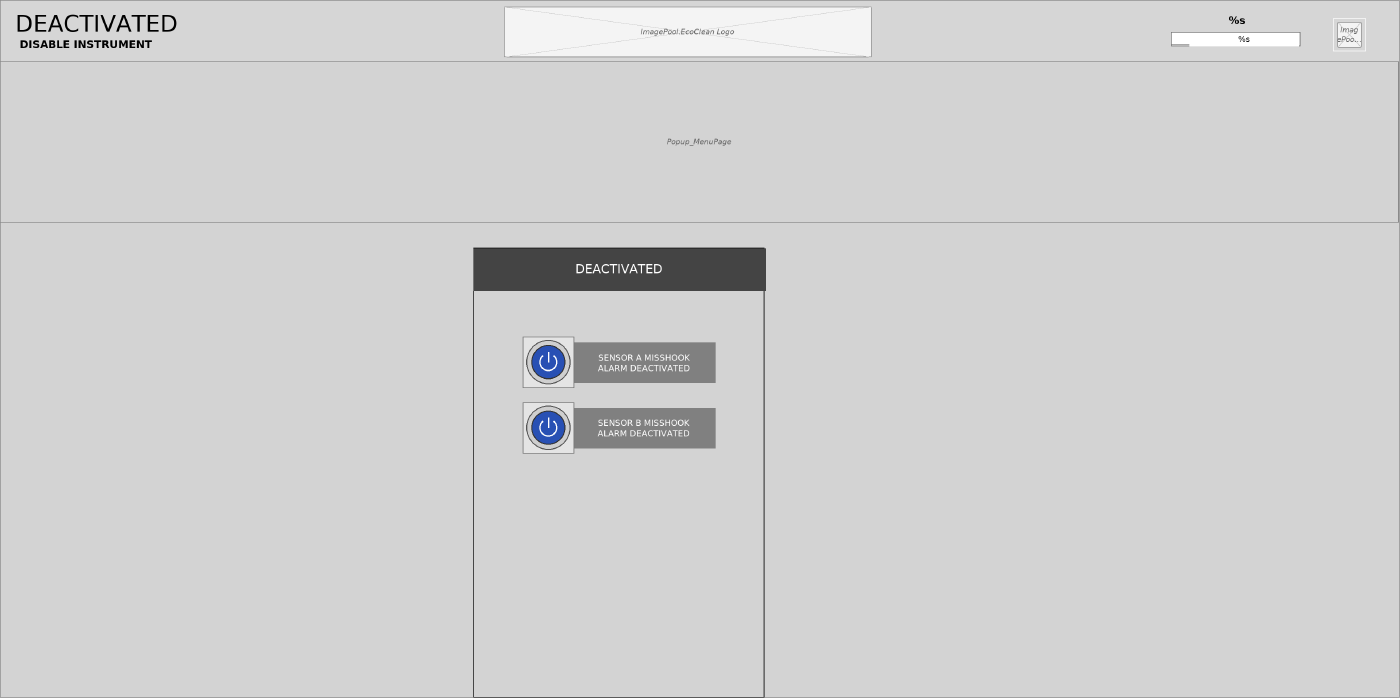
VISUALIZATION Deactivated_Page  // 1920x958
    Rectangle (0,63 1920x26)
        p3528305787: HMI_Ctrl.ANIMATION3
    Rectangle (0,0 1919x85)
    Label (18,6 267x53), "DEACTIVATED"
    Label (24,49 320x24), "DISABLE INSTRUMENT"
    Frame (0,84 1918x221), invisible if: HMI_Ctrl.CloseMenuButton
        shows Popup_MenuPage()
    Group (1828,25 45x45)
        OnMouseClick: toggle HMI_Ctrl.MenuButton
        RoundedRectangle (0,0 45x45), colour toggle: HMI_Ctrl.MenuButton
        Image (6,5 33x35), image: ImagePool.Menu Button
    Rectangle (649,340 399x618)
    Rectangle (649,341 401x58)
    Label (786,357 274x24), "DEACTIVATED"
    RoundedRectangle (766,470 215x55)
    Label (789,473 189x51), "SENSOR A MISSHOOK ALARM DEACTIVATED"
    PowerSwitch (717,462 70x70), variable: ARbArmMissHookByPass1[1], behaviour: TOGGLE, style: Switch-PowerSwitch-Blue
    RoundedRectangle (766,560 215x55)
    Label (788,563 190x50), "SENSOR B MISSHOOK ALARM DEACTIVATED"
    PowerSwitch (717,552 70x70), variable: ARbArmMissHookByPass2[1], behaviour: TOGGLE, style: Switch-PowerSwitch-Blue
    Image (691,9 504x69), image: ImagePool.EcoClean Logo
    Group (1606,17 179x46)
        Button (0,27 177x19), image: VisuSymbols.Symbols.AddUser
        Rectangle (25,28 150x18), "%s", text variable: fbHmiTF1800_UserlevelManagement.dsHmiUserStatus_Active.sLoginName
        Rectangle (2,0 177x22), "%s", text variable: DSLocalSystemTimeML.sCurrentDT24Hr_General
END_VISUALIZATION

(* stored: Version 1.1.0.1, ProductVersion 3.1.4024.12
   Visu Deactivated_Page: Id {f0df98f5-20cd-4493-845a-8ffa9bc7a8c4} *)
